(* CODESYS project Portal Manual Operation.project

Project tree, tasks and I/O mapping:
  Device : CODESYS Control for Raspberry Pi, 3S - Smart Software Solutions GmbH, version 3.5.11.20
    application Application
      libraries: Standard, * (System); Util, * (System); VisuDialogs, * (System)
      task MainTask (cyclic, interval 4 ms, priority 1) calls PLC_PRG
      task Profinet_IOTask (cyclic, interval t#1ms, priority 1) calls nothing
      task Profinet_CommunicationTask (cyclic, interval t#10ms, priority 30) calls PN_Controller.CommCycle
      task VISU_TASK (cyclic, interval 100 ms, priority 31) calls VisuElems.Visu_Prg
      program PLC_PRG [CFC]
      function block PortalAnsteuerung [ST]
      data type Position
      data type TwoByteOverInteger
      function block Handbetrieb [ST]
      visualisation Visualization
      function block AnimationSteuerung [ST]
      function block RfidBedienung [ST]
    SoftMotion General Axis Pool
    I²C
    SPI
    GPIOs_A_B : GPIOs A/B, 3S - Smart Software Solutions GmbH, version 3.5.11.0
        unmapped channels: digital inputs (GPIO0..GPIO31), digital outputs (GPIO0..GPIO31)
    Onewire
    Camera device
      <Leer>
    Ethernet : Ethernet, 3S - Smart Software Solutions GmbH, version 3.5.11.0
        settings: IPAddress = [192,168,24,190]; SubnetMask = [255,255,255,0]; GatewayAddress = [192,168,24,1]; MACAddress = [16#B8,16#27,16#EB,16#AD,16#CF,16#C6]; NetworkInterfaceName = 'eth0'; NetworkInterfaceName = "eth0"; SaveCommunicationSettings = FALSE
      PN_Controller : PN-Controller, 3S - Smart Software Solutions GmbH, order no. 1, version 3.5.11.30
          settings: First IP Address = [192, 168, 24, 225]; Last IP Address = [192, 168, 24, 225]; Default Subnet Mask = [255, 255, 255, 0]; Default Gateway Address = [0, 0, 0, 0]; PDPortDataCheck.PeerStationName = ''
        Portal : Portal, BBS Brinkstraße, order no. 6ES7 214-1AG40-0XB0, version SW=V4.2, HW=
            settings: Slave parameters.Identification.IP address = [192,168,24,225]; Slave parameters.Identification.Subnet mask = [255,255,255,0]; Slave parameters.Identification.Default gateway = [0,0,0,0]; Slave parameters.Identification.MAC address = [16#00,16#00,16#00,16#00,16#00,16#00]; Slave parameters.Identification.Station name = 'portal6'; Slave parameters.Reduction ratio = 16; Slave parameters.Watchdog interval = 15; swapInfoOutputs = [10,6,7,5,10,1,2,15]; swapInfoInputs = [10,6,7,5,2,16]; swapInfoOutputs = [10,2,2,126]; swapInfoInputs = [10,2,2,126]; PDPortDataCheck.PeerStationName = ''
            output Application.PLC_PRG.LedStart : BOOL  // Outputs.Portal In Panel.LED Start
            output Application.PLC_PRG.LedReset : BOOL  // Outputs.Portal In Panel.LED Reset
            output Application.PLC_PRG.MotorenAktivieren : BOOL  // Outputs.Portal In Control.Motoren einschalten
            output Application.PLC_PRG.GreiferOeffnenPN : BOOL  // Outputs.Portal In Control.Greifer öffnen
            output Application.PLC_PRG.GreiferSchliessenPN : BOOL  // Outputs.Portal In Control.Greifer schließen
            output Application.PLC_PRG.StartHoming : BOOL  // Outputs.Portal In Move.Referenzfahrt starten
            output Application.PLC_PRG.StartPositionierungXY : BOOL  // Outputs.Portal In Move.Positionierung XY starten
            output Application.PLC_PRG.StartPositionierungZ : BOOL  // Outputs.Portal In Move.Positionierung Z starten
            output Application.PLC_PRG.SollPositionX : INT  // Outputs.Position X (0,1 mm)
            output Application.PLC_PRG.SollPositionY : INT  // Outputs.Position Y (0,1 mm)
            output Application.PLC_PRG.SollPositionZ : INT  // Outputs.Position Z (0,1 mm)
            input  Application.PLC_PRG.StartButton : BOOL  // Inputs.Portal Out Panel.Button Start
            input  Application.PLC_PRG.StopButton : BOOL  // Inputs.Portal Out Panel.Button Stop
            input  Application.PLC_PRG.ResetButton : BOOL  // Inputs.Portal Out Panel.Button Reset
            input  Application.PLC_PRG.MotorenAktiv : BOOL  // Inputs.Portal Out Control State.Motoren eingeschaltet
            input  Application.PLC_PRG.GreiferAuf : BOOL  // Inputs.Portal Out Control State.Greifer offen
            input  Application.PLC_PRG.GreiferZu : BOOL  // Inputs.Portal Out Control State.Greifer geschlossen
            input  Application.PLC_PRG.HomingFertig : BOOL  // Inputs.Portal Out Move State.Referenzfahrt fertig
            input  Application.PLC_PRG.PositionXYFertig : BOOL  // Inputs.Portal Out Move State.Positionierung XY fertig
            input  Application.PLC_PRG.PositionZFertig : BOOL  // Inputs.Portal Out Move State.Positionierung Z fertig
            input  Application.PLC_PRG.IstPositionX : INT  // Inputs.Position X (0,1 mm)
            input  Application.PLC_PRG.IstPositionY : INT  // Inputs.Position Y (0,1 mm)
            input  Application.PLC_PRG.IstPositionZ : INT  // Inputs.Position Z (0,1 mm)
            output Application.PLC_PRG.LesenStarten : BOOL  // Outputs.Rfid In Control.Lesen starten
            output Application.PLC_PRG.SchreibenStarten : BOOL  // Outputs.Rfid In Control.Schreiben starten
            output Application.PLC_PRG.SchreibDaten  // Outputs.RfidIn
            input  Application.PLC_PRG.TagVorhanden : BOOL  // Inputs.Rfid Out Control.Tag vorhanden
            input  Application.PLC_PRG.RfidFertig : BOOL  // Inputs.Rfid Out Control.RFID fertig
            input  Application.PLC_PRG.LeseDaten  // Inputs.RfidOut
            unmapped channels: Outputs, Inputs, Outputs, Inputs
  text list GlobalTextList
*)

// Device/Application/Position
TYPE Position :
STRUCT
	X: INT;
	Y: INT;
	Z: INT;
END_STRUCT
END_TYPE

// Device/Application/TwoByteOverInteger
TYPE TwoByteOverInteger :
UNION
	i: INT;
	bytes: ARRAY [0..1] OF BYTE;
END_UNION
END_TYPE

// Device/Application/PLC_PRG
PROGRAM PLC_PRG
VAR
	PortalAnsteuerung_1: PortalAnsteuerung;
	Handbetrieb_0: Handbetrieb;
	ZielPositionX: INT;
	ZielPositionY: INT;
	ZielPositionZ: INT;
	GreiferZu: BOOL;
	GreiferAuf: BOOL;
	GreiferSchliessen: BOOL;
	GreiferOeffnen: BOOL;
	startFahrt: BOOL;
	startReferenzFahrt: BOOL;
	AnimationSteuerung_0: AnimationSteuerung;
	MotorenAktiv: BOOL;
	HomingFertig: BOOL;
	PositionZFertig: BOOL;
	PositionXYFertig: BOOL;
	IstPositionX: INT;
	IstPositionY: INT;
	IstPositionZ: INT;
	MotorenAktivieren: BOOL;
	StartHoming: BOOL;
	SollPositionX: INT := 500;
	SollPositionY: INT := 3000;
	SollPositionZ: INT := 450;
	StartPositionierungZ: BOOL;
	StartPositionierungXY: BOOL;
	StartButton: BOOL;
	StopButton: BOOL;
	ResetButton: BOOL;
	LedStart: BOOL;
	LedReset: BOOL;
	temp: INT;
	RfidIn: ARRAY[0..127] OF BYTE;
	tempRfidIn: ARRAY[0..127] OF BYTE;
	LeseDaten: ARRAY [0..125] OF BYTE;
	SchreibDaten: ARRAY [0..125] OF BYTE;
	RfidBedienung_0: RfidBedienung;
	TagVorhanden: BOOL;
	RfidFertig: BOOL;
	StarteLesen: BOOL;
	StarteSchreiben: BOOL;
	LesenStarten: BOOL;
	SchreibenStarten: BOOL;
	GreiferOeffnenPN: BOOL;
	GreiferSchliessenPN: BOOL;
END_VAR

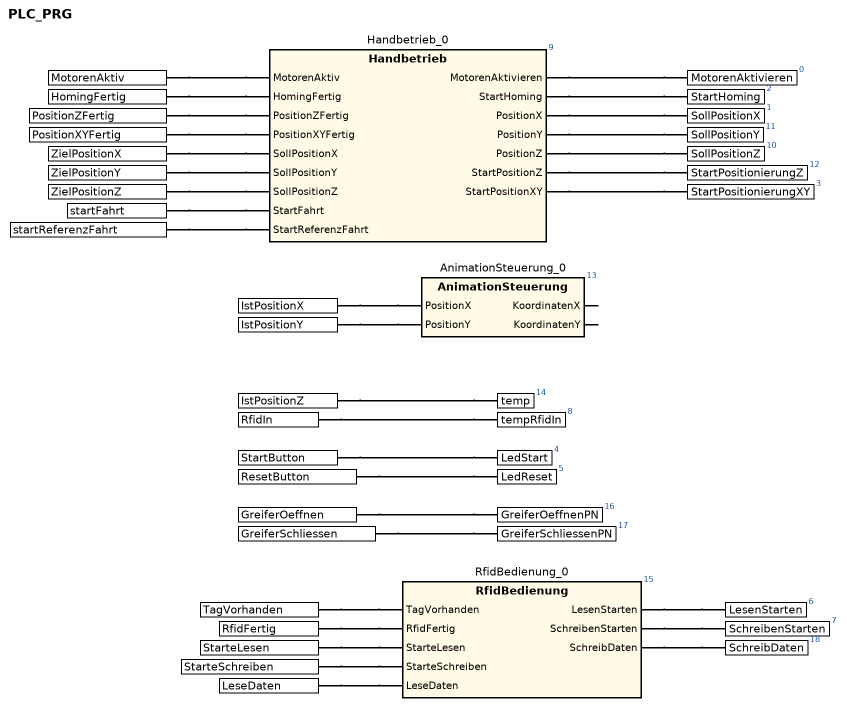
// note: 5 stored wires end on pins the file does not list and are not shown
MotorenAktivieren := Handbetrieb_0.MotorenAktivieren;
SollPositionX := Handbetrieb_0.PositionX;
StartHoming := Handbetrieb_0.StartHoming;
StartPositionierungXY := Handbetrieb_0.StartPositionXY;
LedStart := StartButton;
LedReset := ResetButton;
LesenStarten := RfidBedienung_0.LesenStarten;
SchreibenStarten := RfidBedienung_0.SchreibenStarten;
tempRfidIn := RfidIn;
Handbetrieb_0(
    MotorenAktiv := MotorenAktiv,
    HomingFertig := HomingFertig,
    PositionZFertig := PositionZFertig,
    PositionXYFertig := PositionXYFertig,
    SollPositionX := ZielPositionX,
    SollPositionY := ZielPositionY,
    SollPositionZ := ZielPositionZ,
    StartFahrt := startFahrt,
    StartReferenzFahrt := startReferenzFahrt); // Handbetrieb
SollPositionZ := Handbetrieb_0.PositionZ;
SollPositionY := Handbetrieb_0.PositionY;
StartPositionierungZ := Handbetrieb_0.StartPositionZ;
AnimationSteuerung_0(PositionX := IstPositionX, PositionY := IstPositionY); // AnimationSteuerung
temp := IstPositionZ;
RfidBedienung_0(
    TagVorhanden := TagVorhanden,
    RfidFertig := RfidFertig,
    StarteLesen := StarteLesen,
    StarteSchreiben := StarteSchreiben,
    LeseDaten := LeseDaten); // RfidBedienung
GreiferOeffnenPN := GreiferOeffnen;
GreiferSchliessenPN := GreiferSchliessen;
SchreibDaten := RfidBedienung_0.SchreibDaten;

END_PROGRAM

// Device/Application/Handbetrieb
FUNCTION_BLOCK Handbetrieb
VAR_INPUT
	MotorenAktiv: BOOL;
	HomingFertig: BOOL;
	PositionZFertig: BOOL;
	PositionXYFertig: BOOL;
	SollPositionX: INT;
	SollPositionY: INT;
	SollPositionZ: INT;
	StartFahrt: BOOL;
	StartReferenzFahrt: BOOL;
END_VAR
VAR_OUTPUT
	MotorenAktivieren: BOOL;
	StartHoming: BOOL;
	PositionX: INT;
	PositionY: INT;
	PositionZ: INT;
	StartPositionZ: BOOL;
	StartPositionXY: BOOL;
END_VAR
VAR
	iStep: INT;
END_VAR


CASE iStep OF
	
    0:
        MotorenAktivieren := TRUE;
		iStep := 10;
		
    10:
        IF MotorenAktiv THEN
            StartHoming := TRUE;
            iStep := 20;
        END_IF;

    20:
        IF HomingFertig THEN
            StartHoming := FALSE;
            iStep := 100;
        END_IF;

	100:
        IF StartFahrt THEN
            iStep := 200;
        END_IF;
		
		IF StartReferenzFahrt THEN
            iStep := 10;
        END_IF;
	
	
    200:
	    // Starte Fahrt in Z-Richtung
        PositionZ := SollPositionZ;
        StartPositionZ := TRUE;

        IF PositionZFertig THEN
            StartPositionZ := FALSE;	
            iStep := 210;
        END_IF;

    210:
	    // Starte Fahrt in XY-Richtung
		PositionX := SollPositionX;
        PositionY := SollPositionY;
        StartPositionXY := TRUE;

        IF PositionXYFertig THEN
            StartPositionXY := FALSE;
            iStep := 100;
        END_IF;

END_CASE;

END_FUNCTION_BLOCK

// Device/Application/AnimationSteuerung
FUNCTION_BLOCK AnimationSteuerung
VAR_INPUT
	PositionX: INT;
	PositionY: INT;
END_VAR
VAR_OUTPUT
	KoordinatenX: INT;
	KoordinatenY: INT;
END_VAR
VAR
END_VAR


KoordinatenX := (PositionX / 10);
KoordinatenY := 390 - (PositionY / 10);

END_FUNCTION_BLOCK

// Device/Application/RfidBedienung
FUNCTION_BLOCK RfidBedienung
VAR_INPUT
	TagVorhanden: BOOL;
	RfidFertig: BOOL;
	StarteLesen: BOOL;
	StarteSchreiben: BOOL;
	LeseDaten: ARRAY [0..125] OF BYTE;
END_VAR
VAR_OUTPUT
	LesenStarten: BOOL;
	SchreibenStarten: BOOL;
	SchreibDaten: ARRAY [0..125] OF BYTE;
END_VAR
VAR
	StartTaster: BOOL;
	StartFlanke: R_TRIG;
END_VAR


StartFlanke(CLK:=StarteLesen OR StarteSchreiben);

IF StartFlanke.Q AND StarteLesen AND TagVorhanden THEN
	LesenStarten := TRUE;
END_IF;

IF NOT StarteLesen THEN
	LesenStarten := FALSE;
END_IF;

IF StartFlanke.Q AND StarteSchreiben AND TagVorhanden THEN
	SchreibenStarten := TRUE;
END_IF;

IF NOT StarteSchreiben THEN
	SchreibenStarten := FALSE;
END_IF;

SchreibDaten[1] := 142;
SchreibDaten[2] := 77;
SchreibDaten[3] := 255;

END_FUNCTION_BLOCK

// Device/Application/PortalAnsteuerung
FUNCTION_BLOCK PortalAnsteuerung
VAR_INPUT
	StopButton: BOOL;
	ResetButton: BOOL;
	MotorenAktiv: BOOL;
	HomingFertig: BOOL;
	StartButton: BOOL;
	PositionZFertig: BOOL;
	PositionXYFertig: BOOL;
END_VAR
VAR_OUTPUT
	MotorenAktivieren: BOOL;
	StartHoming: BOOL;
	PositionX: INT;
	PositionY: INT;
	PositionZ: INT;
	StartPositionZ: BOOL;
	StartPositionXY: BOOL;
	LedStart: BOOL;
	LedReset: BOOL;
END_VAR
VAR
	PosT1: Position;
	iStep: INT;
	n: INT;
	delay: TON;
	blinker: Blink;
END_VAR


//  ##################  wichtige Koordinaten
PosT1.X := 600; //760;   // Erste Probe
PosT1.Y := 2250; //2250;
PosT1.Z := 100;

// LED in Tastern blinken lassen
blinker(enable:=TRUE, timehigh:=T#0.5S, timelow:=T#0.5S);
LedStart := (iStep > 100) OR (iStep = 100 AND blinker.OUT);
LedReset := (iStep = 30) OR (iStep = 10 AND blinker.OUT);

IF NOT StopButton THEN
    iStep := 0;
END_IF;

CASE iStep OF
	
    0:
        iStep := 10;
        // ######## Grundstellung anfahren ###########   

    10:
        IF ResetButton THEN 
            MotorenAktivieren := TRUE;
            iStep := 20;
        END_IF;

    20:
        IF MotorenAktiv THEN
            StartHoming := TRUE;
            iStep := 30;
        END_IF;

    30:
        IF HomingFertig THEN
            StartHoming := FALSE;
            iStep := 100;
        END_IF;

        // ######## Automatik Start ###########   

    100:
        // Greifer schließen
        //"PN_SimulationIn".Aktoren.MB5 := false;
        //"PN_SimulationIn".Aktoren.MB6 := true;

        IF ResetButton THEN
            iStep := 20;
        END_IF;

        IF StartButton THEN
            n := 0;
            PositionX := PosT1.X;
            PositionY := PosT1.Y;

            iStep := 200;
        END_IF;

        // ######## Postitionierung Pipette ########  

    200:
        PositionZ := 500;
        StartPositionZ := TRUE;

        IF PositionZFertig THEN
            StartPositionZ := FALSE;
            PositionX := PositionX + 250;
            PositionY := PositionY + 25;
			
            iStep := 210;
        END_IF;

    210:
        PositionZ := PosT1.Z;
        StartPositionXY := TRUE;

        IF PositionXYFertig THEN
            StartPositionXY := FALSE;
			
            iStep := 220;
        END_IF;
       
    220:
        StartPositionZ := TRUE;

        IF PositionZFertig THEN
            StartPositionZ := FALSE;
			
            delay(IN := TRUE, PT := T#500MS);

            IF delay.Q THEN
                delay(IN := FALSE, PT := T#500MS);

                iStep := 230;
            END_IF;
        END_IF;

    230:
        n := n + 1;

        IF n < 4 THEN
            iStep := 200;
        ELSE
            iStep := 100;
        END_IF;

END_CASE;

END_FUNCTION_BLOCK

// Device/Application/Visualization
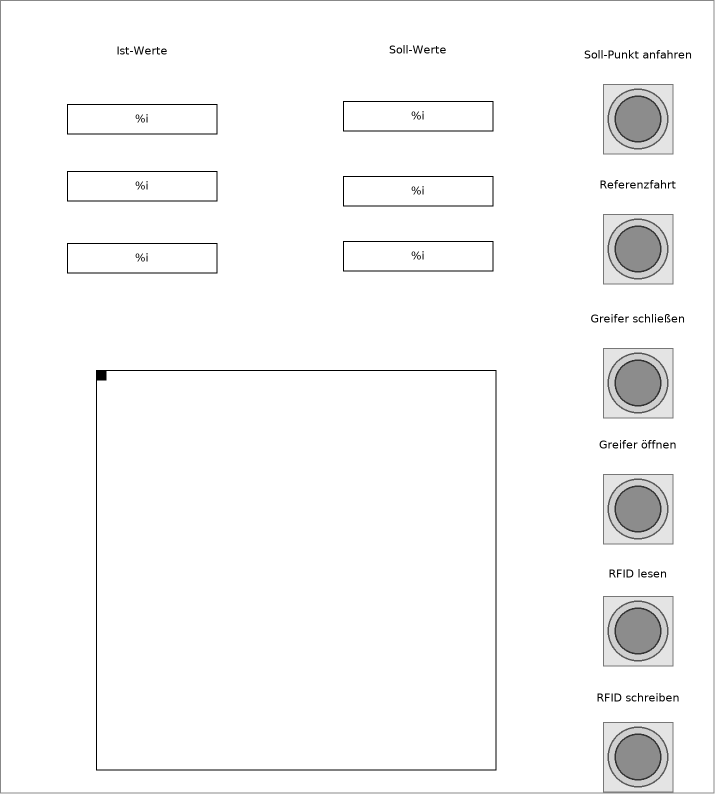
VISUALIZATION Visualization  // 715x794
    Rectangle (67,104 150x30), "%i", text variable: PLC_PRG.IstPositionX
    Rectangle (67,171 150x30), "%i", text variable: PLC_PRG.IstPositionY
    Rectangle (67,243 150x30), "%i", text variable: PLC_PRG.IstPositionZ
    Rectangle (343,101 150x30), "%i", text variable: PLC_PRG.ZielPositionX
        OnMouseDown: write the text variable via Default, min 0, max 3900
    Rectangle (343,176 150x30), "%i", text variable: PLC_PRG.ZielPositionY
        OnMouseDown: write the text variable via Default, min 0, max 3900
    Rectangle (343,241 150x30), "%i", text variable: PLC_PRG.ZielPositionZ
        OnMouseDown: write the text variable via Default, min 0, max 470
    Rectangle (67,36 150x30), "Ist-Werte"
    Rectangle (343,35 150x30), "Soll-Werte"
    PushSwitch (603,84 70x70), variable: PLC_PRG.startFahrt, behaviour: TAP, style: Switch-PushSwitch-Gray
    Rectangle (563,40 150x30), "Soll-Punkt anfahren"
    PushSwitch (603,214 70x70), variable: PLC_PRG.startReferenzFahrt, behaviour: TAP, style: Switch-PushSwitch-Gray
    Rectangle (563,170 150x30), "Referenzfahrt"
    Rectangle (96,370 400x400)
    Rectangle (96,370 10x10)
        p874137650: PLC_PRG.AnimationSteuerung_0.KoordinatenX
        p1126004900: PLC_PRG.AnimationSteuerung_0.KoordinatenY
        p3528305787: PLC_PRG.AnimationSteuerung_0.KoordinatenX
        p2773130477: PLC_PRG.AnimationSteuerung_0.KoordinatenY
    PushSwitch (603,348 70x70), variable: PLC_PRG.GreiferSchliessen, behaviour: TAP, style: Switch-PushSwitch-Gray
    Rectangle (563,304 150x30), "Greifer schließen"
    PushSwitch (603,474 70x70), variable: PLC_PRG.GreiferOeffnen, behaviour: TAP, style: Switch-PushSwitch-Gray
    Rectangle (563,430 150x30), "Greifer öffnen"
    PushSwitch (603,596 70x70), variable: PLC_PRG.StarteLesen, behaviour: TAP, style: Switch-PushSwitch-Gray
    Rectangle (563,559 150x30), "RFID lesen"
    PushSwitch (603,722 70x70), variable: PLC_PRG.StarteSchreiben, behaviour: TAP, style: Switch-PushSwitch-Gray
    Rectangle (563,683 150x30), "RFID schreiben"
END_VISUALIZATION
